FUNCTION_BLOCK FB_GenerateData
VAR_INPUT
	bRun			: BOOL;
	pDataStructure	: POINTER TO ST_TemperatureStructure;
END_VAR
VAR_OUTPUT
END_VAR
VAR
	fbGetSystemTime	: GETSYSTEMTIME;
END_VAR

fbGetSystemTime();
IF(bRun)THEN
	IF(pDataStructure <>0)THEN
		pDataStructure^.fRoomTemperature		:= 21 + pDataStructure^.fRoomTemperature * SIN(fbGetSystemTime.timeLoDW);
		pDataStructure^.fBathRoomTemperature	:= 18 + pDataStructure^.fBathRoomTemperature * COS(fbGetSystemTime.timeLoDW);
		pDataStructure^.diSomeOtherData			:= pDataStructure^.diSomeOtherData + (DWORD_TO_DINT(fbGetSystemTime.timeLoDW));
	END_IF
END_IF

END_FUNCTION_BLOCK

(* stored: Version 1.1.0.1, ProductVersion 3.1.4024.3
   POU FB_GenerateData: Id {4f21bb5e-b102-4330-81b9-65413e0613d3}, SpecialFunc None *)
